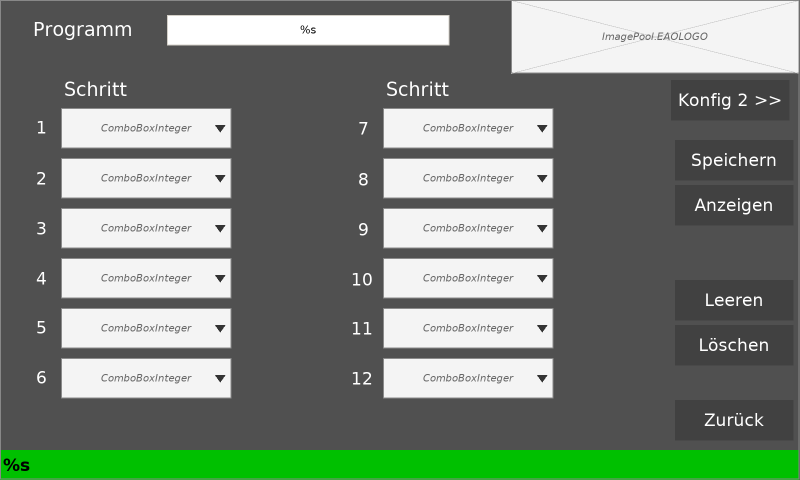
VISUALIZATION Konfig1  // 800x480
    Image (511,0 288x73), image: ImagePool.EAOLOGO
    Textfield (30,15 200x29), "Programm"
    Rectangle (0,450 799x30), "%s", text variable: MAIN.HMI.sStatus, colour variable: MAIN.HMI.nColorInfoBalken
        p3450524324: MAIN.HMI.nColorInfoBalken
    RoundedRectangle (675,325 118x40), "Löschen"
        OnMouseClick: execute { MAIN.HMI.bBtnProgrammLoeschen := TRUE; }
    ComboBoxInteger (61,108 170x40), variable: MAIN.HMI.ProgrammTemp.aAktorBew[1].nNummer, text list: 'TL_Aktoren'
    Textfield (167,15 282x30), "%s", text variable: MAIN.HMI.ProgrammTemp.sName
        OnMouseClick: write the text variable via VisuDialogs.Keypad
    RoundedRectangle (675,140 118x40), "Speichern", colour toggle: MAIN.fbWritePersistentData.BUSY
        OnMouseClick: execute { MAIN.HMI.bBtnProgrammSpeichern := TRUE; }
    RoundedRectangle (675,185 118x40), "Anzeigen"
        OnMouseClick: execute { MAIN.HMI.bBtnProgrammAnzeigen := TRUE; }
    ComboBoxInteger (61,158 170x40), variable: MAIN.HMI.ProgrammTemp.aAktorBew[2].nNummer, text list: 'TL_Aktoren'
    ComboBoxInteger (61,208 170x40), variable: MAIN.HMI.ProgrammTemp.aAktorBew[3].nNummer, text list: 'TL_Aktoren'
    ComboBoxInteger (61,258 170x40), variable: MAIN.HMI.ProgrammTemp.aAktorBew[4].nNummer, text list: 'TL_Aktoren'
    ComboBoxInteger (61,308 170x40), variable: MAIN.HMI.ProgrammTemp.aAktorBew[5].nNummer, text list: 'TL_Aktoren'
    ComboBoxInteger (61,358 170x40), variable: MAIN.HMI.ProgrammTemp.aAktorBew[6].nNummer, text list: 'TL_Aktoren'
    Textfield (61,75 139x29), "Schritt"
    RoundedRectangle (671,80 118x40), "Konfig 2 >>"
        OnMouseClick: change screen: Konfig2
    Textfield (383,75 156x29), "Schritt"
    ComboBoxInteger (383,108 170x40), variable: MAIN.HMI.ProgrammTemp.aAktorBew[7].nNummer, text list: 'TL_Aktoren'
    ComboBoxInteger (383,158 170x40), variable: MAIN.HMI.ProgrammTemp.aAktorBew[8].nNummer, text list: 'TL_Aktoren'
    ComboBoxInteger (383,208 170x40), variable: MAIN.HMI.ProgrammTemp.aAktorBew[9].nNummer, text list: 'TL_Aktoren'
    ComboBoxInteger (383,258 170x40), variable: MAIN.HMI.ProgrammTemp.aAktorBew[10].nNummer, text list: 'TL_Aktoren'
    ComboBoxInteger (383,308 170x40), variable: MAIN.HMI.ProgrammTemp.aAktorBew[11].nNummer, text list: 'TL_Aktoren'
    ComboBoxInteger (383,358 170x40), variable: MAIN.HMI.ProgrammTemp.aAktorBew[12].nNummer, text list: 'TL_Aktoren'
    RoundedRectangle (675,280 118x40), "Leeren"
        OnMouseClick: execute { MAIN.HMI.bBtnKonfigLeeren := TRUE; }
    RoundedRectangle (675,400 118x40), "Zurück"
        OnMouseClick: change screen: Zyklusbetrieb
    Textfield (33,113 34x29), "1"
    Textfield (33,214 34x29), "3"
    Textfield (33,264 34x29), "4"
    Textfield (33,164 34x29), "2"
    Textfield (33,313 34x29), "5"
    Textfield (33,363 34x29), "6"
    Textfield (355,114 34x29), "7"
    Textfield (355,215 34x29), "9"
    Textfield (348,265 34x29), "10"
    Textfield (355,165 34x29), "8"
    Textfield (348,314 34x29), "11"
    Textfield (348,364 34x29), "12"
    Group (800,90 645x290)
        RoundedRectangle (0,0 645x290), "%s", text variable: MAIN.HMI.sPopUpText, colour toggle: MAIN.fbWritePersistentData.BUSY, invisible if: NOT MAIN.HMI.bPopUpAnzeigen
            p3560616238: MAIN.HMI.nPopUpXOffset
        RoundedRectangle (128,197 118x40), "Ja", colour toggle: MAIN.fbWritePersistentData.BUSY, invisible if: NOT MAIN.HMI.bPopUpAnzeigen
            p3560616238: MAIN.HMI.nPopUpXOffset
            OnMouseClick: execute { MAIN.HMI.bBtnPopUpJa := TRUE; }
        RoundedRectangle (405,198 118x40), "Nein", colour toggle: MAIN.fbWritePersistentData.BUSY, invisible if: NOT MAIN.HMI.bPopUpAnzeigen
            p3560616238: MAIN.HMI.nPopUpXOffset
            OnMouseClick: execute { MAIN.HMI.bBtnPopUpNein := TRUE; }
END_VISUALIZATION

(* stored: Version 1.1.0.1, ProductVersion 3.1.4024.12
   Visu Konfig1: Id {e2481534-9345-4843-b01a-66aeb67aea7e} *)
